// TIA Portal V17 export
// export: Created 2022-12-08T07:31:25.8530917Z, ExportSetting WithDefaults, DisplayName Totally Integrated Automation Portal, DisplayVersion V17 Update 5, DisplayName TIA Portal Openness, DisplayVersion V17 Update 5, DisplayName TIA Portal Version Control Interface, DisplayVersion V17, DisplayName Simotion SCOUT TIA, DisplayVersion 5.4.3.0, DisplayName SINAMICS Startdrive Advanced, DisplayVersion V17 SP1, DisplayName SINAMICS Startdrive G130, G150, S120, S150, SINAMICS MV, S210, DisplayVersion V17 SP1, DisplayName SINAMICS Startdrive G110M, G120, G120C, G120D, G120P, G115D, DisplayVersion V17 SP1, DisplayName STEP 7 Professional, DisplayVersion V17 Update 5, DisplayName STEP 7 Safety, DisplayVersion V17, DisplayName WinCC Advanced, DisplayVersion V17 Update 5
FUNCTION_BLOCK "FB_BDE"   // FB700, FBD
{ S7_Optimized_Access := 'TRUE' }
AUTHOR : EconoPak GmbH
VERSION : 0.1
// stored: AutoNumber true, IsIECCheckEnabled true, IsRetainMemResEnabled false, MemoryReserve 100, SetENOAutomatically true, UDAEnableTagReadback false
   VAR_INPUT
      i_CountTotal_OK : DInt;   // Zähleingang für Produkte in Ordnung / Counting input for products alright / Laskentatulo tuotteille, jotka ovat kunnossa / Entrée de compteur pour les produits corrects / Tellende ingang voor producten in orde / Wejście zliczające dla produktów w porządku / Счетчик ввод для продуктов в порядке / Entrada de recuento para productos correctos
      i_CountTotal_NOK : DInt;   // Zähleingang für Produkte nicht Ordnung / Counting input for products not all right / Laskentatulo tuotteille ei ole kunnossa / Entrée de compteur pour les produits pas bien / Tellende ingang voor producten niet in orde / Wejście zliczające dla produktów nie w porządku / Счетчики для продуктов не в порядке / Entrada de recuento para productos no bien
      i_CountTotal_In : DInt;   // Zähleingang für Produkte Erkannt / Counting input for products Detected / Laskentatulo tuotteille Havaitut tuotteet / Entrée de compteur pour les produits détectés / Tellende ingang voor producten gedetecteerd / Wejście zliczające dla produktów wykrytych / Счетчик ввод для обнаруженных продуктов / Entrada de recuento para productos detectados
   END_VAR
   VAR_OUTPUT
      q_ProductionData : "UDT_BDE";
   END_VAR
   VAR_IN_OUT
      iq_InformationMessages : "UDT_Messages";
      iq_OperateMessages : "UDT_Messages";
      iq_FaultMessagesAbsolut : "UDT_Messages";
      iq_FaultMessagesCycleEnd : "UDT_Messages";
      iq_OMACGlobalData : "UDT_OMAC_GlobalData";
   END_VAR
   VAR DB_SPECIFIC
      stat_InformationMessages : "UDT_Messages";
   END_VAR
   VAR
      "stat_AT_ InformationMessages" AT stat_InformationMessages : Array[1..256] of Bool;
   END_VAR
   VAR DB_SPECIFIC
      stat_OperateMessages : "UDT_Messages";
   END_VAR
   VAR
      stat_AT_OperateMessages AT stat_OperateMessages : Array[1..256] of Bool;
   END_VAR
   VAR DB_SPECIFIC
      stat_FaultMessagesAbsolut : "UDT_Messages";
   END_VAR
   VAR
      stat_AT_FaultMessagesAbsolut AT stat_FaultMessagesAbsolut : Array[1..256] of Bool;
   END_VAR
   VAR DB_SPECIFIC
      stat_FaultMessagesCycleEnd : "UDT_Messages";
   END_VAR
   VAR
      stat_AT_FaultMessagesCycleEnd AT stat_FaultMessagesCycleEnd : Array[1..256] of Bool;
   END_VAR
   VAR_TEMP
      temp_Counter : Int;
      temp_FaultCodeInformationMessages : Int;
      temp_FaultCodeOperateMessages : Int;
      temp_FaultCodeAbsolut : Int;
      temp_FaultcodeCycleEnd : Int;
   END_VAR
BEGIN

REGION Network 1 (SCL): Mappen der Fehlermeldungen auf interne Variablen
   #stat_FaultMessagesAbsolut    := #iq_FaultMessagesAbsolut;
   #stat_FaultMessagesCycleEnd   := #iq_FaultMessagesCycleEnd;
   #stat_OperateMessages         := #iq_OperateMessages;
   #stat_InformationMessages     := #iq_InformationMessages;
END_REGION

REGION Network 2 (SCL): Fehlercodes generieren
   (/*Eine Hinweismeldung ist akitv*/)
   FOR #temp_Counter := 1 TO 256 BY 1 DO
       IF #"stat_AT_ InformationMessages"[#temp_Counter]
       THEN
           #temp_FaultCodeInformationMessages := #temp_Counter;
           EXIT;
       END_IF;
   END_FOR;
   #q_ProductionData.FaultCodeInformationMessages := #temp_FaultCodeInformationMessages;

   (/*Eine Betriebsmeldung ist akitv*/)
   FOR #temp_Counter := 1 TO 256 BY 1 DO
       IF #stat_AT_OperateMessages[#temp_Counter]
       THEN
           #temp_FaultCodeOperateMessages := #temp_Counter;
           EXIT;
       END_IF;
   END_FOR;
   #q_ProductionData.FaultCodeOperateMessages := #temp_FaultCodeOperateMessages;

   (/*Eine Störmeldung Stop Absolut ist aktiv*/)
   FOR #temp_Counter := 1 TO 256 BY 1 DO
       IF #stat_AT_FaultMessagesAbsolut[#temp_Counter]
       THEN
           #temp_FaultCodeAbsolut := #temp_Counter;
           EXIT;
       END_IF;
   END_FOR;
   #q_ProductionData.FaultCodeFaultMessagesAbsolut := #temp_FaultCodeAbsolut;

   (/*Eine Störmeldung Stop Taktende ist aktiv*/)
   FOR #temp_Counter := 1 TO 256 BY 1 DO
       IF #stat_AT_FaultMessagesCycleEnd[#temp_Counter]
       THEN
           #temp_FaultcodeCycleEnd := #temp_Counter;
           EXIT;
       END_IF;
   END_FOR;
   #q_ProductionData.FaultCodeFaultMessagesCycleEnd := #temp_FaultcodeCycleEnd;
END_REGION

REGION Network 3 (SCL): OMAC mappen
   #q_ProductionData.ActualOMACMode := #iq_OMACGlobalData.UnitModeCurrent;
   #q_ProductionData.ActualOMACStatus := #iq_OMACGlobalData.StateCurrent;
END_REGION

REGION Network 4 (SCL): Produktionszähler mappen
   #q_ProductionData.ProductCountOK := #i_CountTotal_OK;
   #q_ProductionData.ProductCountNOK := #i_CountTotal_NOK;
   #q_ProductionData.ProductCountGesamt := #i_CountTotal_In;
END_REGION
END_FUNCTION_BLOCK
